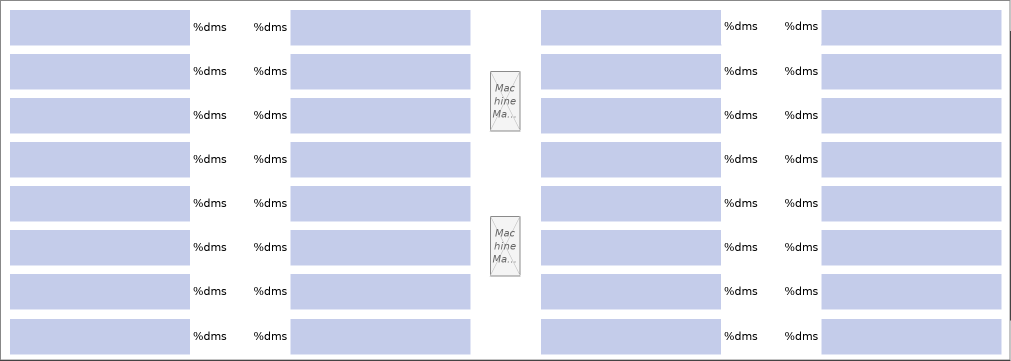
VISUALIZATION CtrlInput  // 1011x361
VAR_INPUT
	In:						POINTER TO BOOL;
	SizeIn:					DINT;
	Enable:					BOOL;// 是否启用强制功能
	Ton:					POINTER TO UINT;// 延迟区域
	In_S:					POINTER TO BOOL;
END_VAR
VAR
	_pageCount:				INT;
	_index:					INT;
END_VAR
    RoundedRectangle (0,0 1010x115)
    RoundedRectangle (0,246 1010x115)
    Rectangle (0,52 1010x268)
    Line (1010,31) (1010,320)
    Line (0,33) (0,332)
    Image (490,71 30x60), image: MachineManage.ImagePool.prev
        OnMouseDown: execute {
            IF _index-32>=0 THEN
            	_index:=_index-32;
            END_IF
        }
    Image (490,216 30x60), image: MachineManage.ImagePool.next
        OnMouseClick: execute {
            IF SizeIn>_index+32 THEN
            	_index:=_index+32;
            END_IF
        }
    RoundedRectangle (10,10 180x35), colour toggle: In[_index], invisible if: SizeIn<=_index, input disabled if: In_S[_index], text list: 'InputText', text index: _index
        OnMouseClick: execute {
            IF Enable AND SizeIn>_index THEN
            	In[_index]:=NOT In[_index];
            END_IF;
        }
    RoundedRectangle (10,54 180x35), colour toggle: In[1+_index], invisible if: SizeIn<= 1+_index, input disabled if: In_S[1+_index], text list: 'InputText', text index: 1+_index
        OnMouseClick: execute {
            IF Enable AND SizeIn>_index+1 THEN
            	In[_index+1]:=NOT In[_index+1];
            END_IF;
        }
    RoundedRectangle (10,98 180x35), colour toggle: In[2+_index], invisible if: SizeIn<= 2+_index, input disabled if: In_S[2+_index], text list: 'InputText', text index: 2+_index
        OnMouseClick: execute {
            IF Enable AND SizeIn>_index+2 THEN
            	In[_index+2]:=NOT In[_index+2];
            END_IF;
        }
    RoundedRectangle (10,142 180x35), colour toggle: In[3+_index], invisible if: SizeIn<=3+_index, input disabled if: In_S[3+_index], text list: 'InputText', text index: 3+_index
        OnMouseClick: execute {
            IF Enable AND SizeIn>_index+3 THEN
            	In[_index+3]:=NOT In[_index+3];
            END_IF;
        }
    RoundedRectangle (10,186 180x35), colour toggle: In[_index+4], invisible if: SizeIn<=_index+4, input disabled if: In_S[_index+4], text list: 'InputText', text index: _index+4
        OnMouseClick: execute {
            IF Enable AND SizeIn>_index+4 THEN
            	In[_index+4]:=NOT In[_index+4];
            END_IF;
        }
    RoundedRectangle (10,230 180x35), colour toggle: In[_index+5], invisible if: SizeIn<=_index+5, input disabled if: In_S[_index+5], text list: 'InputText', text index: _index+5
        OnMouseClick: execute {
            IF Enable AND SizeIn>_index+5 THEN
            	In[_index+5]:=NOT In[_index+5];
            END_IF;
        }
    RoundedRectangle (10,274 180x35), colour toggle: In[_index+6], invisible if: SizeIn<=_index+6, input disabled if: In_S[_index+6], text list: 'InputText', text index: _index+6
        OnMouseClick: execute {
            IF Enable AND SizeIn>_index+6 THEN
            	In[_index+6]:=NOT In[_index+6];
            END_IF;
        }
    RoundedRectangle (10,319 180x35), colour toggle: In[_index+7], invisible if: SizeIn<=_index+7, input disabled if: In_S[_index+7], text list: 'InputText', text index: _index+7
        OnMouseClick: execute {
            IF Enable AND SizeIn>_index+7 THEN
            	In[_index+7]:=NOT In[_index+7];
            END_IF;
        }
    RoundedRectangle (290,10 180x35), colour toggle: In[_index+8], invisible if: SizeIn<=_index+8, input disabled if: In_S[_index+8], text list: 'InputText', text index: _index+8
        OnMouseClick: execute {
            IF Enable AND SizeIn>_index+8 THEN
            	In[_index+8]:=NOT In[_index+8];
            END_IF;
        }
    RoundedRectangle (290,54 180x35), colour toggle: In[_index+9], invisible if: SizeIn<=_index+9, input disabled if: In_S[_index+9], text list: 'InputText', text index: _index+9
        OnMouseClick: execute {
            IF Enable AND SizeIn>_index+9 THEN
            	In[_index+9]:=NOT In[_index+9];
            END_IF;
        }
    RoundedRectangle (290,98 180x35), colour toggle: In[_index+10], invisible if: SizeIn<=_index+10, input disabled if: In_S[_index+10], text list: 'InputText', text index: _index+10
        OnMouseClick: execute {
            IF Enable AND SizeIn>_index+10 THEN
            	In[_index+10]:=NOT In[_index+10];
            END_IF;
        }
    RoundedRectangle (290,142 180x35), colour toggle: In[_index+11], invisible if: SizeIn<=_index+11, input disabled if: In_S[_index+11], text list: 'InputText', text index: _index+11
        OnMouseClick: execute {
            IF Enable AND SizeIn>_index+11 THEN
            	In[_index+11]:=NOT In[_index+11];
            END_IF;
        }
    RoundedRectangle (290,186 180x35), colour toggle: In[_index+12], invisible if: SizeIn<=_index+12, input disabled if: In_S[_index+12], text list: 'InputText', text index: _index+12
        OnMouseClick: execute {
            IF Enable AND SizeIn>_index+12 THEN
            	In[_index+12]:=NOT In[_index+12];
            END_IF;
        }
    RoundedRectangle (290,230 180x35), colour toggle: In[_index+13], invisible if: SizeIn<=_index+13, input disabled if: In_S[_index+13], text list: 'InputText', text index: _index+13
        OnMouseClick: execute {
            IF Enable AND SizeIn>_index+13 THEN
            	In[_index+13]:=NOT In[_index+13];
            END_IF;
        }
    RoundedRectangle (290,274 180x35), colour toggle: In[_index+14], invisible if: SizeIn<=_index+14, input disabled if: In_S[_index+14], text list: 'InputText', text index: _index+14
        OnMouseClick: execute {
            IF Enable AND SizeIn>_index+14 THEN
            	In[_index+14]:=NOT In[_index+14];
            END_IF;
        }
    RoundedRectangle (290,319 180x35), colour toggle: In[_index+15], invisible if: SizeIn<=_index+15, input disabled if: In_S[_index+15], text list: 'InputText', text index: _index+15
        OnMouseClick: execute {
            IF Enable AND SizeIn>_index+15 THEN
            	In[_index+15]:=NOT In[_index+15];
            END_IF;
        }
    RoundedRectangle (541,10 180x35), colour toggle: In[_index+16], invisible if: SizeIn<=_index+16, input disabled if: In_S[_index+16], text list: 'InputText', text index: _index+16
        OnMouseClick: execute {
            IF Enable AND SizeIn>_index+16 THEN
            	In[_index+16]:=NOT In[_index+16];
            END_IF;
        }
    RoundedRectangle (541,54 180x35), colour toggle: In[_index+17], invisible if: SizeIn<=_index+17, input disabled if: In_S[_index+17], text list: 'InputText', text index: _index+17
        OnMouseClick: execute {
            IF Enable AND SizeIn>_index+17 THEN
            	In[_index+17]:=NOT In[_index+17];
            END_IF;
        }
    RoundedRectangle (541,98 180x35), colour toggle: In[_index+18], invisible if: SizeIn<=_index+18, input disabled if: In_S[_index+18], text list: 'InputText', text index: _index+18
        OnMouseClick: execute {
            IF Enable AND SizeIn>_index+18 THEN
            	In[_index+18]:=NOT In[_index+18];
            END_IF;
        }
    RoundedRectangle (541,142 180x35), colour toggle: In[_index+19], invisible if: SizeIn<=_index+19, input disabled if: In_S[_index+19], text list: 'InputText', text index: _index+19
        OnMouseClick: execute {
            IF Enable AND SizeIn>_index+19 THEN
            	In[_index+19]:=NOT In[_index+19];
            END_IF;
        }
    RoundedRectangle (541,186 180x35), colour toggle: In[_index+20], invisible if: SizeIn<=_index+20, input disabled if: In_S[_index+20], text list: 'InputText', text index: _index+20
        OnMouseClick: execute {
            IF Enable AND SizeIn>_index+20 THEN
            	In[_index+20]:=NOT In[_index+20];
            END_IF;
        }
    RoundedRectangle (541,230 180x35), colour toggle: In[_index+21], invisible if: SizeIn<=_index+21, input disabled if: In_S[_index+21], text list: 'InputText', text index: _index+21
        OnMouseClick: execute {
            IF Enable AND SizeIn>_index+21 THEN
            	In[_index+21]:=NOT In[_index+21];
            END_IF;
        }
    RoundedRectangle (541,274 180x35), colour toggle: In[_index+22], invisible if: SizeIn<=_index+22, input disabled if: In_S[_index+22], text list: 'InputText', text index: _index+22
        OnMouseClick: execute {
            IF Enable AND SizeIn>_index+22 THEN
            	In[_index+22]:=NOT In[_index+22];
            END_IF;
        }
    RoundedRectangle (541,319 180x35), colour toggle: In[_index+23], invisible if: SizeIn<=_index+23, input disabled if: In_S[_index+23], text list: 'InputText', text index: _index+23
        OnMouseClick: execute {
            IF Enable AND SizeIn>_index+23 THEN
            	In[_index+23]:=NOT In[_index+23];
            END_IF;
        }
    RoundedRectangle (821,10 180x35), colour toggle: In[_index+24], invisible if: SizeIn<=_index+24, input disabled if: In_S[_index+24], text list: 'InputText', text index: _index+24
        OnMouseClick: execute {
            IF Enable AND SizeIn>_index+24 THEN
            	In[_index+24]:=NOT In[_index+24];
            END_IF;
        }
    RoundedRectangle (821,54 180x35), colour toggle: In[_index+25], invisible if: SizeIn<=_index+25, input disabled if: In_S[_index+25], text list: 'InputText', text index: _index+25
        OnMouseClick: execute {
            IF Enable AND SizeIn>_index+25 THEN
            	In[_index+25]:=NOT In[_index+25];
            END_IF;
        }
    RoundedRectangle (821,98 180x35), colour toggle: In[_index+26], invisible if: SizeIn<=_index+26, input disabled if: In_S[_index+26], text list: 'InputText', text index: _index+26
        OnMouseClick: execute {
            IF Enable AND SizeIn>_index+26 THEN
            	In[_index+26]:=NOT In[_index+26];
            END_IF;
        }
    RoundedRectangle (821,142 180x35), colour toggle: In[_index+27], invisible if: SizeIn<=_index+27, input disabled if: In_S[_index+27], text list: 'InputText', text index: _index+27
        OnMouseClick: execute {
            IF Enable AND SizeIn>_index+27 THEN
            	In[_index+27]:=NOT In[_index+27];
            END_IF;
        }
    RoundedRectangle (821,186 180x35), colour toggle: In[_index+28], invisible if: SizeIn<=_index+28, input disabled if: In_S[_index+28], text list: 'InputText', text index: _index+28
        OnMouseClick: execute {
            IF Enable AND SizeIn>_index+28 THEN
            	In[_index+28]:=NOT In[_index+28];
            END_IF;
        }
    RoundedRectangle (821,230 180x35), colour toggle: In[_index+29], invisible if: SizeIn<=_index+29, input disabled if: In_S[_index+29], text list: 'InputText', text index: _index+29
        OnMouseClick: execute {
            IF Enable AND SizeIn>_index+29 THEN
            	In[_index+29]:=NOT In[_index+29];
            END_IF;
        }
    RoundedRectangle (821,274 180x35), colour toggle: In[_index+30], invisible if: SizeIn<=_index+30, input disabled if: In_S[_index+30], text list: 'InputText', text index: _index+30
        OnMouseClick: execute {
            IF Enable AND SizeIn>_index+30 THEN
            	In[_index+30]:=NOT In[_index+30];
            END_IF;
        }
    RoundedRectangle (821,319 180x35), colour toggle: In[_index+31], invisible if: SizeIn<=_index+31, input disabled if: In_S[_index+31], text list: 'InputText', text index: _index+31
        OnMouseClick: execute {
            IF Enable AND SizeIn>_index+31 THEN
            	In[_index+31]:=NOT In[_index+31];
            END_IF;
        }
    Rectangle (190,10 50x35), "%dms", text variable: Ton[_index], invisible if: SizeIn<=_index
        OnMouseClick: write the text variable via Default, min 0
    Rectangle (240,10 50x35), "%dms", text variable: Ton[_index+8], invisible if: SizeIn<=_index+8
        OnMouseClick: write the text variable via Default, min 0
    Rectangle (190,54 50x35), "%dms", text variable: Ton[_index+1], invisible if: SizeIn<=_index+1
        OnMouseClick: write the text variable via Default, min 0
    Rectangle (240,54 50x35), "%dms", text variable: Ton[_index+9], invisible if: SizeIn<=_index+9
        OnMouseClick: write the text variable via Default, min 0
    Rectangle (190,98 50x35), "%dms", text variable: Ton[_index+2], invisible if: SizeIn<=_index+2
        OnMouseClick: write the text variable via Default, min 0
    Rectangle (240,98 50x35), "%dms", text variable: Ton[_index+10], invisible if: SizeIn<=_index+10
        OnMouseClick: write the text variable via Default, min 0
    Rectangle (190,142 50x35), "%dms", text variable: Ton[_index+3], invisible if: SizeIn<=_index+3
        OnMouseClick: write the text variable via Default, min 0
    Rectangle (240,142 50x35), "%dms", text variable: Ton[_index+11], invisible if: SizeIn<=_index+11
        OnMouseClick: write the text variable via Default, min 0
    Rectangle (190,186 50x35), "%dms", text variable: Ton[_index+4], invisible if: SizeIn<=_index+4
        OnMouseClick: write the text variable via Default, min 0
    Rectangle (240,186 50x35), "%dms", text variable: Ton[_index+12], invisible if: SizeIn<=_index+12
        OnMouseClick: write the text variable via Default, min 0
    Rectangle (190,230 50x35), "%dms", text variable: Ton[_index+5], invisible if: SizeIn<=_index+5
        OnMouseClick: write the text variable via Default, min 0
    Rectangle (240,230 50x35), "%dms", text variable: Ton[_index+13], invisible if: SizeIn<=_index+13
        OnMouseClick: write the text variable via Default, min 0
    Rectangle (190,274 50x35), "%dms", text variable: Ton[_index+6], invisible if: SizeIn<=_index+6
        OnMouseClick: write the text variable via Default, min 0
    Rectangle (240,274 50x35), "%dms", text variable: Ton[_index+14], invisible if: SizeIn<=_index+14
        OnMouseClick: write the text variable via Default, min 0
    Rectangle (190,319 50x35), "%dms", text variable: Ton[_index+7], invisible if: SizeIn<=_index+7
        OnMouseClick: write the text variable via Default, min 0
    Rectangle (240,319 50x35), "%dms", text variable: Ton[_index+15], invisible if: SizeIn<=_index+15
        OnMouseClick: write the text variable via Default, min 0
    Rectangle (721,9 50x35), "%dms", text variable: Ton[_index+16], invisible if: SizeIn<=_index+16
        OnMouseClick: write the text variable via Default, min 0
    Rectangle (771,9 50x35), "%dms", text variable: Ton[_index+24], invisible if: SizeIn<=_index+24
        OnMouseClick: write the text variable via Default, min 0
    Rectangle (721,54 50x35), "%dms", text variable: Ton[_index+17], invisible if: SizeIn<=_index+17
        OnMouseClick: write the text variable via Default, min 0
    Rectangle (771,54 50x35), "%dms", text variable: Ton[_index+25], invisible if: SizeIn<=_index+25
        OnMouseClick: write the text variable via Default, min 0
    Rectangle (721,98 50x35), "%dms", text variable: Ton[_index+18], invisible if: SizeIn<=_index+18
        OnMouseClick: write the text variable via Default, min 0
    Rectangle (771,98 50x35), "%dms", text variable: Ton[_index+26], invisible if: SizeIn<=_index+26
        OnMouseClick: write the text variable via Default, min 0
    Rectangle (721,142 50x35), "%dms", text variable: Ton[_index+19], invisible if: SizeIn<=_index+19
        OnMouseClick: write the text variable via Default, min 0
    Rectangle (771,142 50x35), "%dms", text variable: Ton[_index+27], invisible if: SizeIn<=_index+27
        OnMouseClick: write the text variable via Default, min 0
    Rectangle (721,186 50x35), "%dms", text variable: Ton[_index+20], invisible if: SizeIn<=_index+20
        OnMouseClick: write the text variable via Default, min 0
    Rectangle (771,186 50x35), "%dms", text variable: Ton[_index+28], invisible if: SizeIn<=_index+28
        OnMouseClick: write the text variable via Default, min 0
    Rectangle (721,230 50x35), "%dms", text variable: Ton[_index+21], invisible if: SizeIn<=_index+21
        OnMouseClick: write the text variable via Default, min 0
    Rectangle (771,230 50x35), "%dms", text variable: Ton[_index+29], invisible if: SizeIn<=_index+29
        OnMouseClick: write the text variable via Default, min 0
    Rectangle (721,274 50x35), "%dms", text variable: Ton[_index+22], invisible if: SizeIn<=_index+22
        OnMouseClick: write the text variable via Default, min 0
    Rectangle (771,274 50x35), "%dms", text variable: Ton[_index+30], invisible if: SizeIn<=_index+30
        OnMouseClick: write the text variable via Default, min 0
    Rectangle (721,319 50x35), "%dms", text variable: Ton[_index+23], invisible if: SizeIn<=_index+23
        OnMouseClick: write the text variable via Default, min 0
    Rectangle (771,319 50x35), "%dms", text variable: Ton[_index+31], invisible if: SizeIn<=_index+31
        OnMouseClick: write the text variable via Default, min 0
END_VISUALIZATION

(* stored: Version 1.1.0.1, ProductVersion 3.1.4024.3
   Visu CtrlInput: Id {36242466-fbd9-4352-8ed4-f1ecb5f844c6} *)
